TYPE "UDT_TIME_PLANTA"
VERSION : 0.1
   STRUCT
      BRITADORES  : "UDT_TIME_BRITADORES";
      TRANSPORTADORES : "UDT_TIME_TRANSPORTADORES";
      PENEIRAS : "UDT_TIME_PENEIRAS";
      CALHAS : "UDT_TIME_CALHAS";
   END_STRUCT;

END_TYPE